(* PLC project Generated.project, CODESYS CODESYS V3.5 SP19 Patch 1 *)
(* stored: creationDateTime 2026-08-22T23:52:43.806205, modificationDateTime 2026-08-22T23:52:43.806205 *)

(* ═══════════════════════════════════════════════════════════════ 🔌 ST_EncoderHw — Frontière hardware codeur (IN/OUT) ─────────────────────────────────────────────────────────────── 🎯 Regroupe les entrées/sorties hardware d'un codeur absolu EtherCAT pour exposer l'interface physique de FB_Encoder de façon testable. 🔌 Producteur/consommateur : PRG_02_Acquisition câble ce bus vers le device. 📄 Doc : DOC/AF/AF_Partie-09_Fonction_Encoder_v2.1.md ═══════════════════════════════════════════════════════════════ *)
TYPE ST_EncoderHw : STRUCT
  RawPosIn : UDINT;  (* === ENTREES BUS ETHERCAT (vers le codeur) === Position brute EtherCAT (in) *)
  AlarmsIn : UINT;  (* Codes alarmes bruts EtherCAT *)
  WarningsIn : UINT;  (* Codes avertissements bruts EtherCAT *)
  SlaveOperational : BOOL;  (* Esclave EtherCAT operationnel *)
  PresetAck : BOOL;  (* Pulse confirmation preset reussi *)
  PresetNak : BOOL;  (* Pulse echec / timeout preset *)
  PresetTriggerCmd : WORD;  (* === SORTIES BUS (vers le codeur) === Ordre declenchement preset vers PDO Rx *)
  CodeSeqTriggerCmd : WORD;  (* Ordre sequence code vers PDO Rx *)
  PresetValueOut : UDINT;  (* Valeur de preset transmise au PDO Rx *)
END_STRUCT;
END_TYPE
